{attribute 'qualified_only'}
{attribute 'strict'}
TYPE schudmachineStatus :
(
	enum_member := 0
);
END_TYPE

(* stored: Version 1.1.0.1, ProductVersion 3.1.4024.15
   DUT schudmachineStatus: Id {888e5b6e-002e-46a4-955b-683faa694f03} *)
